{attribute 'qualified_only'}
VAR_GLOBAL
    // InCmd
    {attribute 'OPC.UA.DA' := '1'}
    {attribute 'OPC.UA.DA.StructuredType' := '1'}
    g_stBigBagMassBalanceInCmd      : ST_BigBagMassBalanceInCmd;

    // Par
    {attribute 'OPC.UA.DA' := '1'}
    {attribute 'OPC.UA.DA.StructuredType' := '1'}
    g_stBigBagMassBalancePar        : ST_BigBagMassBalancePar;

    // InValues
    {attribute 'OPC.UA.DA' := '1'}
    {attribute 'OPC.UA.DA.StructuredType' := '1'}
    g_stBigBagMassBalanceInValues   : ST_BigBagMassBalanceInValues;

    // Status
    {attribute 'OPC.UA.DA' := '1'}
    {attribute 'OPC.UA.DA.StructuredType' := '1'}
    g_stBigBagMassBalanceStatus     : ST_BigBagMassBalanceStatus;

    // OutValues
    {attribute 'OPC.UA.DA' := '1'}
    {attribute 'OPC.UA.DA.StructuredType' := '1'}
    g_stBigBagMassBalanceOutValues  : ST_BigBagMassBalanceOutValues;
END_VAR

(* stored: Version 1.1.0.1, ProductVersion 3.1.4024.16
   GVL GVL_BigBagMassBalance: Id {66071858-2323-45de-894e-b6f169177c84} *)
